// TIA Portal project "P1_Ejercicio3" (V15.1)

(* hardware
DEVICE "S7-1200 station_1"  S7-1200 Station
   slot 0: "Rack_0"  S7-1200 Rack  Rack  V1.0
   slot 1: "PLC_1"  CPU 1215C AC/DC/Rly  6ES7 215-1BG40-0XB0  V4.2
DEVICE "HMI_1"  KTP900 Basic PN
   slot 0: "HMI_1"  KTP900 Basic PN  6AV2 123-2JB03-0AX0  15.1.0.0
   slot 1: "HMI_RT_1"  KTP900 Basic PN  6AV2 123-2JB03-0AX0  15.1.0.0
   slot 5: "HMI_1.IE_CP_1"  PROFINET Interface  15.0.1.0
      slot 1: "Interfaz PROFINET_1"  PROFINET Interface
         slot 1: "Port_1"  Port
*)

// ===== PLC "PLC_1"  CPU 1215C AC/DC/Rly =====

VAR_GLOBAL   // PLC tag table "Tabla de variables estándar"
   "Pulsador de marcha" AT %M0.0 : Bool;
   "Pulsador de paro" AT %M0.1 : Bool;
   "1.Pila de pales en la entrada" AT %M0.2 : Bool;
   "2.Pila de pales en desapilador" AT %M0.3 : Bool;
   "3.Palé en rodillos de salida" AT %M0.4 : Bool;
   "4.Cilindro subir pila pales reposo" AT %M0.5 : Bool;
   "5.Cilindro subir pila pales arriba" AT %M0.6 : Bool;
   "6.Cilindro uña sujetar pila reposo" AT %M0.7 : Bool;
   "7.Cilindro uña sujetar pila extendida" AT %M1.0 : Bool;
   "8.Freno pila recogido" AT %M1.1 : Bool;
   "9.Freno pila extendido" AT %M1.2 : Bool;
   "M1.Motor rodillos entrada pilas" AT %M10.0 : Bool;
   "M2.Motor rodillos desapilador" AT %M10.1 : Bool;
   "M3.Motor rodillos salida de palé" AT %M10.2 : Bool;
   "C1.Cilindro subir pila" AT %M10.3 : Bool;
   "C2.Cilindro uñas sujetar pila" AT %M10.4 : Bool;
   "C3.Cilindro freno" AT %M10.5 : Bool;
   "paletaEn2?" AT %M2.0 : Bool;
   "paletaListaParaSalir" AT %M2.1 : Bool;
   "Permiso_extraer_pale" AT %M1.3 : Bool;
   "sin_permiso" AT %M1.4 : Bool;
   "aux1" AT %M1.5 : Bool;
   "aux2" AT %M1.6 : Bool;
   "c2 desactivado" AT %M1.7 : Bool;
END_VAR

// folder: System blocks/Program resources

DATA_BLOCK "temporizador 3s"   // DB1
{ S7_Optimized_Access := 'TRUE' }
AUTHOR : Simatic
FAMILY : IEC
NAME : IEC_TMR
VERSION : 1.0
// stored: InstanceOfName IEC_TIMER
"IEC_TIMER"
BEGIN
END_DATA_BLOCK

DATA_BLOCK "IEC_Timer_0_DB"   // DB3
{ S7_Optimized_Access := 'TRUE' }
AUTHOR : Simatic
FAMILY : IEC
NAME : IEC_TMR
VERSION : 1.0
// stored: InstanceOfName IEC_TIMER
"IEC_TIMER"
BEGIN
END_DATA_BLOCK

// folder: (top level)

ORGANIZATION_BLOCK "Main"   // OB1, LAD, ProgramCycle
TITLE = "Main Program Sweep (Cycle)" / Ejercicio 3: Control de un desapilador automático.
{ S7_Optimized_Access := 'TRUE' }
VERSION : 0.1
   VAR_INPUT
      Initial_Call : Bool;   // Initial call of this OB
      Remanence : Bool;   // =True, if remanent data are available
   END_VAR
   VAR_TEMP   // added for the SCL form of the ladder/FBD networks
      _w1 : Bool;
      _w2 : Bool;
   END_VAR
BEGIN

REGION Network 1
   // ⬤Tenemos un pulsador de marcha uno de paro para el sistema. Si se pulsa el paro la secuencia se
   // detiene continuando en el mismo punto cuando se pulse marcha de nuevo.
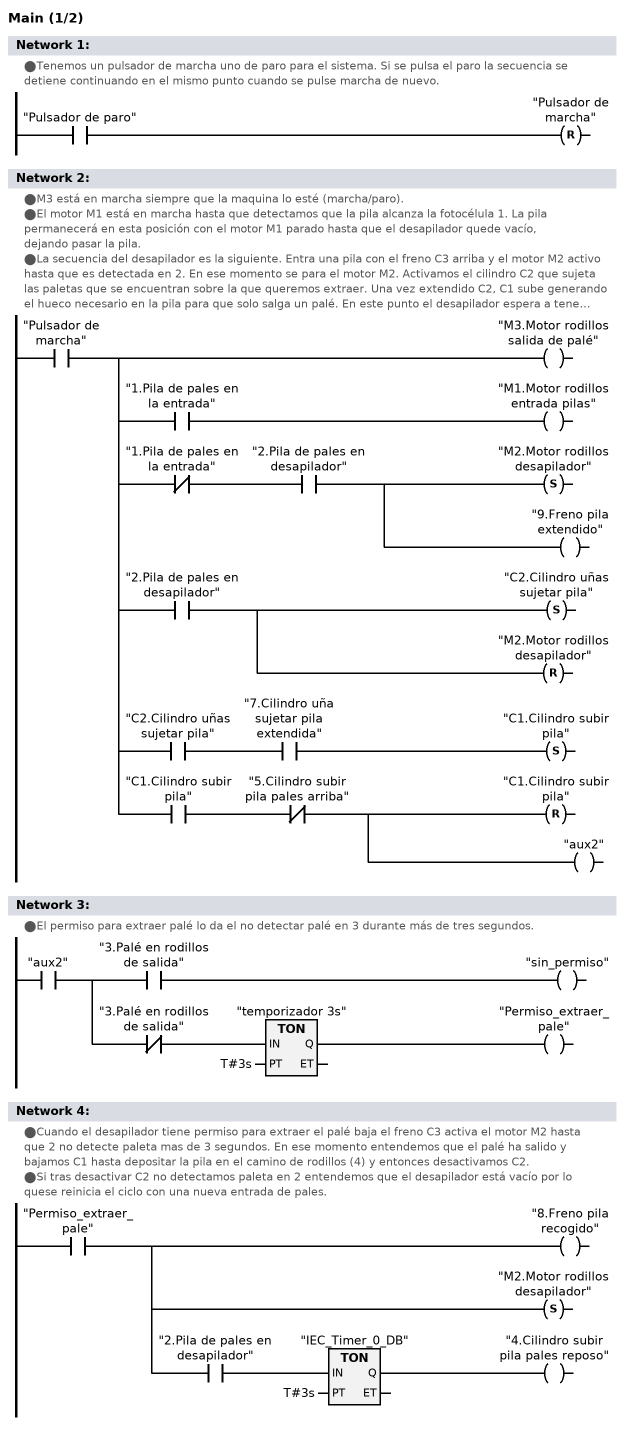
   RUNG wire#powerrail
      Contact( "Pulsador de paro" )
      R_Coil( "Pulsador de marcha" )
   END_RUNG
   // the same network as SCL:
   IF "Pulsador de paro" THEN "Pulsador de marcha" := FALSE; END_IF;
END_REGION

REGION Network 2
   // ⬤M3 está en marcha siempre que la maquina lo esté (marcha/paro). 
   // ⬤El motor M1 está en marcha hasta que detectamos que la pila alcanza la fotocélula 1. La pila
   // permanecerá en esta posición con el motor M1 parado hasta que el desapilador quede vacío,
   // dejando pasar la pila. 
   // ⬤La secuencia del desapilador es la siguiente. Entra una pila con el freno C3 arriba y el motor M2 activo hasta que es detectada en 2. En ese momento se para el motor M2. Activamos el cilindro C2 que sujeta las paletas que se encuentran sobre la que queremos extraer. Una vez extendido C2, C1 sube generando el hueco necesario en la pila para que solo salga un palé. En este punto el desapilador espera a tener permiso para extraer palé.
   RUNG wire#powerrail
      Contact( "Pulsador de marcha" )
      wire#w1
      Coil( "M3.Motor rodillos salida de palé" )
   END_RUNG
   RUNG wire#w1
      Contact( "1.Pila de pales en la entrada" )
      Coil( "M1.Motor rodillos entrada pilas" )
   END_RUNG
   RUNG wire#w1
      I_Contact( "1.Pila de pales en la entrada" )
      Contact( "2.Pila de pales en desapilador" )
      wire#w2
      S_Coil( "M2.Motor rodillos desapilador" )
   END_RUNG
   RUNG wire#w2
      Coil( "9.Freno pila extendido" )
   END_RUNG
   RUNG wire#w1
      Contact( "2.Pila de pales en desapilador" )
      wire#w3
      S_Coil( "C2.Cilindro uñas sujetar pila" )
   END_RUNG
   RUNG wire#w3
      R_Coil( "M2.Motor rodillos desapilador" )
   END_RUNG
   RUNG wire#w1
      Contact( "C2.Cilindro uñas sujetar pila" )
      Contact( "7.Cilindro uña sujetar pila extendida" )
      S_Coil( "C1.Cilindro subir pila" )
   END_RUNG
   RUNG wire#w1
      Contact( "C1.Cilindro subir pila" )
      I_Contact( "5.Cilindro subir pila pales arriba" )
      wire#w4
      R_Coil( "C1.Cilindro subir pila" )
   END_RUNG
   RUNG wire#w4
      Coil( "aux2" )
   END_RUNG
   // the same network as SCL:
   "M3.Motor rodillos salida de palé" := "Pulsador de marcha";
   "M1.Motor rodillos entrada pilas" := "Pulsador de marcha" AND "1.Pila de pales en la entrada";
   #_w1 := "Pulsador de marcha" AND NOT "1.Pila de pales en la entrada" AND "2.Pila de pales en desapilador";
   IF #_w1 THEN "M2.Motor rodillos desapilador" := TRUE; END_IF;
   "9.Freno pila extendido" := #_w1;
   IF "Pulsador de marcha" AND "2.Pila de pales en desapilador" THEN
       "C2.Cilindro uñas sujetar pila" := TRUE;
       "M2.Motor rodillos desapilador" := FALSE;
   END_IF;
   IF "Pulsador de marcha" AND "C2.Cilindro uñas sujetar pila" AND "7.Cilindro uña sujetar pila extendida" THEN
       "C1.Cilindro subir pila" := TRUE;
   END_IF;
   #_w2 := "Pulsador de marcha" AND "C1.Cilindro subir pila" AND NOT "5.Cilindro subir pila pales arriba";
   IF #_w2 THEN "C1.Cilindro subir pila" := FALSE; END_IF;
   "aux2" := #_w2;
END_REGION

REGION Network 3
   // ⬤El permiso para extraer palé lo da el no detectar palé en 3 durante más de tres segundos.
   "sin_permiso" := "aux2" AND "3.Palé en rodillos de salida";
   "temporizador 3s".TON(IN := "aux2" AND NOT "3.Palé en rodillos de salida", PT := T#3s);
   "Permiso_extraer_pale" := "temporizador 3s".Q;
END_REGION

REGION Network 4
   // ⬤Cuando el desapilador tiene permiso para extraer el palé baja el freno C3 activa el motor M2 hasta
   // que 2 no detecte paleta mas de 3 segundos. En ese momento entendemos que el palé ha salido y
   // bajamos C1 hasta depositar la pila en el camino de rodillos (4) y entonces desactivamos C2. 
   // ⬤Si tras desactivar C2 no detectamos paleta en 2 entendemos que el desapilador está vacío por lo quese reinicia el ciclo con una nueva entrada de pales.
   "8.Freno pila recogido" := "Permiso_extraer_pale";
   IF "Permiso_extraer_pale" THEN "M2.Motor rodillos desapilador" := TRUE; END_IF;
   "IEC_Timer_0_DB".TON(IN := "Permiso_extraer_pale" AND "2.Pila de pales en desapilador", PT := T#3s);
   "4.Cilindro subir pila pales reposo" := "IEC_Timer_0_DB".Q;
END_REGION

REGION Network 5
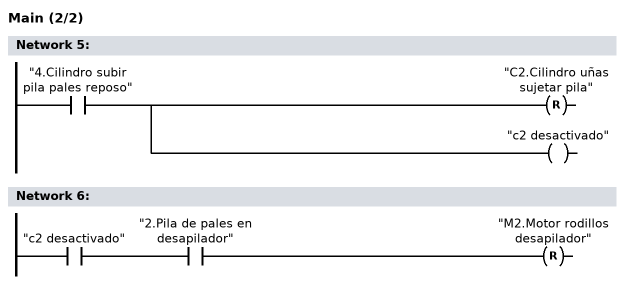
   RUNG wire#powerrail
      Contact( "4.Cilindro subir pila pales reposo" )
      wire#w1
      R_Coil( "C2.Cilindro uñas sujetar pila" )
   END_RUNG
   RUNG wire#w1
      Coil( "c2 desactivado" )
   END_RUNG
   // the same network as SCL:
   IF "4.Cilindro subir pila pales reposo" THEN "C2.Cilindro uñas sujetar pila" := FALSE; END_IF;
   "c2 desactivado" := "4.Cilindro subir pila pales reposo";
END_REGION

REGION Network 6
   RUNG wire#powerrail
      Contact( "c2 desactivado" )
      Contact( "2.Pila de pales en desapilador" )
      R_Coil( "M2.Motor rodillos desapilador" )
   END_RUNG
   // the same network as SCL:
   IF "c2 desactivado" AND "2.Pila de pales en desapilador" THEN
       "M2.Motor rodillos desapilador" := FALSE;
   END_IF;
END_REGION
END_ORGANIZATION_BLOCK

(* ===== HMI "HMI_RT_1" =====
system functions are stored by id; their names below are inferred from use
connection "HMI_Conexión_1": ETHERNET, SMART_S7_1200_OMS

HMI tags "Tabla de variables estándar"
   "Número_imagen_variable" : UInt, internal
   "Pulsador de paro" : Bool = PLC "Pulsador de paro" AT %M0.1, 1 s
   "M1.Motor rodillos entrada pilas" : Bool = PLC "M1.Motor rodillos entrada pilas" AT %M10.0, 1 s
   "M2.Motor rodillos desapilador" : Bool = PLC "M2.Motor rodillos desapilador" AT %M10.1, 1 s
   "M3.Motor rodillos salida de palé" : Bool = PLC "M3.Motor rodillos salida de palé" AT %M10.2, 1 s
   "1.Pila de pales en la entrada" : Bool = PLC "1.Pila de pales en la entrada" AT %M0.2, 1 s
   "2.Pila de pales en desapilador" : Bool = PLC "2.Pila de pales en desapilador" AT %M0.3, 1 s
   "3.Palé en rodillos de salida" : Bool = PLC "3.Palé en rodillos de salida" AT %M0.4, 1 s
   "7.Cilindro uña sujetar pila extendida" : Bool = PLC "7.Cilindro uña sujetar pila extendida" AT %M1.0, 1 s
   "5.Cilindro subir pila pales arriba" : Bool = PLC "5.Cilindro subir pila pales arriba" AT %M0.6, 1 s
   "Pulsador de marcha" : Bool = PLC "Pulsador de marcha" AT %M0.0, 1 s

text list "Nombre_imagen_lista_texto": 1 'Imagen raíz'

Template "Plantilla_1" 800x480
   Button "Salir" at 722,440 size 55x39; TextOff 'Salir'; PictureOff "ExitRuntime_KTP900_Basic_PN_TR"; PictureOn "ExitRuntime_KTP900_Basic_PN_TR"
      on Release: StopRuntime(0)
   Button "Template_Button" at 622,440 size 55x39; TextOff 'Text'
   Button "Template_Button_1" at 522,440 size 55x39; TextOff 'Text'
   Button "Template_Button_2" at 422,440 size 55x39; TextOff 'Text'
   Button "Template_Button_3" at 322,440 size 55x39; TextOff 'Text'
   Button "Template_Button_4" at 222,440 size 55x39; TextOff 'Text'
   Button "Avisos" at 122,440 size 55x39; TextOff 'Avisos'; PictureOff "AlarmDisplay_KTP900_Basic_PN_TR"; PictureOn "AlarmDisplay_KTP900_Basic_PN_TR"
      on Release: function_ef3f5d25("Ventana de avisos_no_acusado", -1)
   Button "Imagen inicial" at 22,440 size 55x39; TextOff 'Imagen inicial'; PictureOff "NavigateHome_KTP900_Basic_PN_TR"; PictureOn "NavigateHome_KTP900_Basic_PN_TR"
      on Release: ActivateScreen("Imagen raíz", 0)
   SymbolicIOField "Imagen_campo_ES_simbólico" at 73,7 size 620x26; TextOff '0'; TextOn '1'; TextList "Nombre_imagen_lista_texto"
      ProcessValue <- "Número_imagen_variable"
      on Change: ActivateScreenByNumber("Número_imagen_variable", 0)
   DateTimeField "HmiScreenItemData" at 695,20 size 105x20
   DateTimeField "HmiScreenItemData_1" at 695,0 size 105x20
   GraphicView "Logotipo" at 0,0 size 71x40; Picture "Logotipo de HMI_1"

screen "Imagen raíz" 800x480, template "Plantilla_1"
   on GenerateScreen: SetTag("Número_imagen_variable", 1)
   Switch "Interruptor_1" at 58,124 size 64x32; CaptionText 'Switch'; TextOff 'OFF'; TextOn 'ON'
      Appearance <- "Pulsador de paro"
      ProcessValue <- "Pulsador de paro"
   TextField "Campo de texto_1" at 67,104 size 41x20; Text 'PARO'
   Switch "Interruptor_2" at 58,179 size 64x32; TextOn 'ON'; CaptionText 'Switch'; TextOff 'OFF'
      ProcessValue <- "Pulsador de marcha"
      Appearance <- "Pulsador de marcha"
   TextField "Campo de texto_2" at 58,159 size 62x20; Text 'MARCHA'
   Switch "Interruptor_3" at 199,96 size 64x32; TextOn 'ON'; CaptionText 'Switch'; TextOff 'OFF'
      ProcessValue <- "1.Pila de pales en la entrada"
      Appearance <- "1.Pila de pales en la entrada"
   TextField "Campo de texto_3" at 146,76 size 173x20; Text '1.Pila de pales en entrada'
   Switch "Interruptor_4" at 199,156 size 64x32; TextOn 'ON'; CaptionText 'Switch'; TextOff 'OFF'
      ProcessValue <- "2.Pila de pales en desapilador"
      Appearance <- "2.Pila de pales en desapilador"
   TextField "Campo de texto_4" at 137,136 size 196x20; Text '2.Pila de pales en desapilador'
   Switch "Interruptor_5" at 206,217 size 64x32; TextOn 'ON'; CaptionText 'Switch'; TextOff 'OFF'
      ProcessValue <- "3.Palé en rodillos de salida"
      Appearance <- "3.Palé en rodillos de salida"
   TextField "Campo de texto_5" at 145,196 size 175x20; Text '3.Palé en rodillos de salida'
   Switch "Interruptor_6" at 432,250 size 64x32; TextOn 'ON'; CaptionText 'Switch'; TextOff 'OFF'
      ProcessValue <- "5.Cilindro subir pila pales arriba"
      Appearance <- "5.Cilindro subir pila pales arriba"
   TextField "Campo de texto_6" at 365,223 size 211x20; Text '5. Cilindro subir pila pales arriba'
   Switch "Interruptor_7" at 434,180 size 64x32; TextOn 'ON'; CaptionText 'Switch'; TextOff 'OFF'
      ProcessValue <- "7.Cilindro uña sujetar pila extendida"
      Appearance <- "7.Cilindro uña sujetar pila extendida"
   TextField "Campo de texto_7" at 353,153 size 237x20; Text '7.Cilindro uña sujetar pila extendida'
   Circle "Círculo_1" at 367,84 size 48x48
      Appearance <- "M1.Motor rodillos entrada pilas"
   TextField "Campo de texto_8" at 365,64 size 56x20; Text 'Motor 1'
   Circle "Círculo_2" at 434,83 size 48x48
      Appearance <- "M2.Motor rodillos desapilador"
   TextField "Campo de texto_9" at 432,63 size 56x20; Text 'Motor 2'
   Circle "Círculo_3" at 508,84 size 48x48
      Appearance <- "M3.Motor rodillos salida de palé"
   TextField "Campo de texto_10" at 506,64 size 56x20; Text 'Motor 3'
*)